FUNCTION alg_a_pusher2 : BOOL
VAR_INPUT
	state: STATE;
END_VAR

alg_a_pusher2 := state.dvar_M_inventory2_a_pusher2;

END_FUNCTION

(* stored: Version 1.1.0.1, ProductVersion 3.1.4022.18
   POU alg_a_pusher2: Id {b641e0de-6a2c-4e6b-b6c8-ffb2fc1e4893}, SpecialFunc None *)
